SUBAPPLICATION tastend (* Subapplication Type *)
  (* Standard: 61499-2; Description: Copyright (c) 2024 Meisterschulen am Ostbahnhof This program and the accompanying materials are made available under the terms of the Eclipse Public License 2.0 which is available at https://www.eclipse.org/legal/epl-2.0/ SPDX-License-Identifier: EPL-2.0 *)
  (* Version 1.0, 2024-10-23, Franz Höpfinger, Meisterschulen am Ostbahnhof *)
  PACKAGE FBs::Uebungen::Uebung_103::subapp;
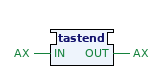
  SOCKETS
    IN : AX;
  END_SOCKETS
  PLUGS
    OUT : AX;
  END_PLUGS
  ADAPTER_CONNECTIONS
    IN TO OUT;
  END_CONNECTIONS
END_SUBAPPLICATION
